Staubli VAL3: listempty.pgx

public program listempty()
  local num lI
  local num lLen
  local string lRun[5]
  local num lRuni
begin
  //
  // Staubli Copyright 2003 06 20
  //
  lLen=size(sItems)-1
  for lI=0 to lLen
    if lI>0
      delete(sItems[0])
      delete(bReadWrite[0])
    endIf
  endFor
  sItems=""
  //
end
